FUNCTION_BLOCK FB_Blink
VAR_INPUT
	OnOffTime : TIME; // Frequency of blinking
	TriggerBlink : BOOL; // If true, blinking is active
END_VAR
VAR_OUTPUT
	BlinkSignal : BOOL; // Turns on/off att set frequency
END_VAR
VAR
	timer1: TON;
	timer2: TON;
END_VAR

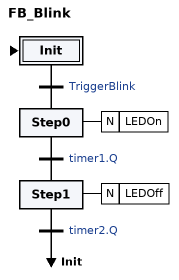
INITIAL_STEP Init:
END_STEP
TRANSITION FROM Init TO Step0
    := TriggerBlink;
END_TRANSITION
STEP Step0:
    LEDOn(N);
END_STEP
TRANSITION FROM Step0 TO Step1
    := timer1.Q;
END_TRANSITION
STEP Step1:
    LEDOff(N);
END_STEP
TRANSITION FROM Step1 TO Init
    := timer2.Q;
END_TRANSITION

ACTION LEDOff:
timer1(IN := FALSE, PT := OnOffTime);
timer2(IN := TRUE, PT := OnOffTime);
BlinkSignal := FALSE;
END_ACTION

ACTION LEDOn:
timer1(IN := TRUE, PT := OnOffTime);
timer2(IN := FALSE, PT := OnOffTime);
BlinkSignal := TRUE;
END_ACTION

END_FUNCTION_BLOCK

(* stored: Version 1.1.0.1, ProductVersion 3.1.4024.13
   POU FB_Blink: Id {adb8d228-e79f-4143-b835-6e6436e7ba2e}, SpecialFunc None
   Action LEDOff: Id {61f2b871-23ee-4f71-aa6b-f618999b3695}
   Action LEDOn: Id {03ef2e14-fe2b-451b-99fd-e5800e271c83} *)
